(* Schneider Machine Expert - Basic project 2. Set and Reset Coil, file version 2.9.0.0 *)
(* ProjectInformations: Name=New project *)

HARDWARE
  Cpu 0: TM221C24R
  EthernetConfiguration: NetworkName=M221, IpAllocationMode=FixedAddress, IpAddress=0.0.0.0, SubnetMask=0.0.0.0
  SerialLineConfiguration: Baud=Baud19200, Parity=ParityEven, DataBits=DataBits8, StopBits=StopBits1, PhysicalMedium=PhysicalMediumRs485, SlaveId=1, Addressing=SlaveAddressing
  MastTask: UsePeriodScanMode=false, PeriodScan=100
  FastTask: Period=255
  CpuBehavior: StartingMode=StartAsPreviousState, AutoSaveRamOnEeprom=true, WatchdogPeriod=250

SYMBOLS  (address, symbol, comment, settings)
  %I0.0     SWITCH_1
  %I0.1     SWITCH_2
  %Q0.0     MOTOR_1

POU New POU
  (* SectionNumber=1 *)

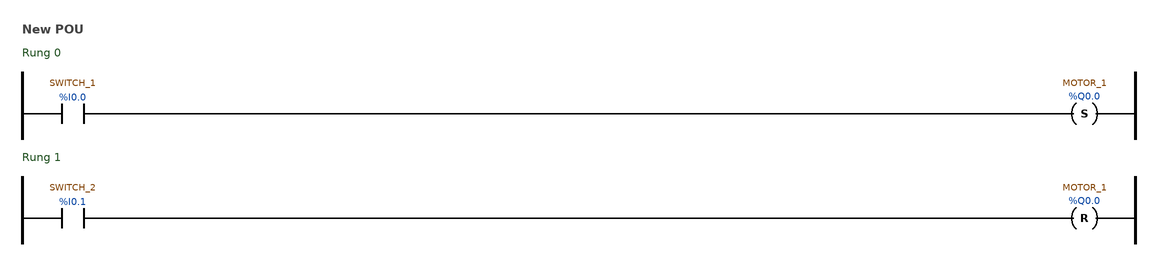

// Rung 0
  LD %I0.0                (* SWITCH_1 *)
  S %Q0.0                 (* MOTOR_1 *)
  // as ST:
  //   IF SWITCH_1 THEN MOTOR_1 := TRUE; END_IF;

// Rung 1
  LD %I0.1                (* SWITCH_2 *)
  R %Q0.0                 (* MOTOR_1 *)
  // as ST:
  //   IF SWITCH_2 THEN MOTOR_1 := FALSE; END_IF;
